// TIA Portal project "CV" (V18)

(* hardware
DEVICE "S7-1500/ET200MP station_1"  S7-1500 station
   slot 0: "Rail_0"  Rack  6ES7 590-1***0-0AA0
   slot 1: "PLC_1"  CPU 1511-1 PN  6ES7 511-1AL03-0AB0  V3.0
      slot 3: "CPU display_1"  6ES7591-1AA00-0AA0
      slot 32768: "PROFINET interface_1"  X1
         slot 32769: "Port_1"  X1 P1
         slot 32770: "Port_2"  X1 P2
      slot 34817: "Virtual CP interface port_1"  Virtual CP interface port  Virtual CP interface port
*)

// ===== PLC "PLC_1"  CPU 1511-1 PN =====

VAR_GLOBAL   // PLC tag table "Default tag table"
   "Tag_1" AT %M0.0 : Bool;
   "Tag_2" AT %Q0.3 : Bool;
   "Tag_3" AT %Q0.4 : Bool;
   "Tag_4" AT %M0.2 : Bool;
   "Tag_5" AT %M0.1 : Bool;
   "Tag_6" AT %Q0.5 : Bool;
   "Tag_7" AT %Q0.6 : Bool;
   "Tag_8" AT %Q0.7 : Bool;
   "Tag_9" AT %Q1.0 : Bool;
END_VAR

ORGANIZATION_BLOCK "Main"   // OB1, LAD, ProgramCycle
TITLE = "Main Program Sweep (Cycle)"
{ S7_Optimized_Access := 'TRUE' }
VERSION : 0.1
   VAR_INPUT
      Initial_Call : Bool;   // Initial call of this OB
      Remanence : Bool;   // =True, if remanent data are available
   END_VAR
BEGIN

REGION Network 1
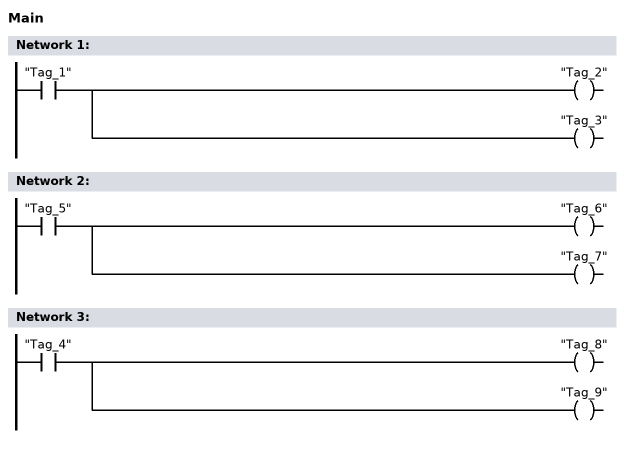
   RUNG wire#powerrail
      Contact( "Tag_1" )
      wire#w1
      Coil( "Tag_2" )
   END_RUNG
   RUNG wire#w1
      Coil( "Tag_3" )
   END_RUNG
   // the same network as SCL:
   "Tag_2" := "Tag_1";
   "Tag_3" := "Tag_1";
END_REGION

REGION Network 2
   RUNG wire#powerrail
      Contact( "Tag_5" )
      wire#w1
      Coil( "Tag_6" )
   END_RUNG
   RUNG wire#w1
      Coil( "Tag_7" )
   END_RUNG
   // the same network as SCL:
   "Tag_6" := "Tag_5";
   "Tag_7" := "Tag_5";
END_REGION

REGION Network 3
   RUNG wire#powerrail
      Contact( "Tag_4" )
      wire#w1
      Coil( "Tag_8" )
   END_RUNG
   RUNG wire#w1
      Coil( "Tag_9" )
   END_RUNG
   // the same network as SCL:
   "Tag_8" := "Tag_4";
   "Tag_9" := "Tag_4";
END_REGION
END_ORGANIZATION_BLOCK